FUNCTION_BLOCK PUBLIC FB_Socket
VAR_OUTPUT
	bActive		: BOOL;
END_VAR

PROPERTY PUBLIC Active : BOOL
GET
Active := bActive;
END_GET
END_PROPERTY

METHOD PUBLIC Off
bActive := false;
END_METHOD

METHOD PUBLIC On
bActive := true;
END_METHOD

END_FUNCTION_BLOCK

(* stored: Version 1.1.0.1, ProductVersion 3.1.4024.12
   POU FB_Socket: Id {6c475d45-e58d-4130-bc0b-b4c64d3e963b}, SpecialFunc None
   Property Active: Id {b49fa6e5-78d3-4844-bf1a-0a8045063ca5}
   Get Get: Id {139bff78-ef9a-42d0-aa93-1fd7fdcb5745}
   Method Off: Id {e36f03c3-37cc-4922-8b54-f1b3d1815351}
   Method On: Id {63e8b64b-b5a9-4311-b930-dda33d9156ba} *)
